PROGRAM program2
VAR
END_VAR

END_PROGRAM

(* stored: Version 1.1.0.1, ProductVersion 3.1.4024.12
   POU program2: Id {cce6f35d-e8e0-431e-8764-77da23c4ebe9}, SpecialFunc None *)
